// TIA Portal V17 export
// export: Created 2023-02-13T11:16:06.1178122Z, ExportSetting WithDefaults, DisplayName Totally Integrated Automation Portal, DisplayVersion V17, DisplayName TIA Portal Openness, DisplayVersion V17, DisplayName TIA Portal Teamcenter Gateway, DisplayVersion V17, DisplayName TIA Portal Version Control Interface, DisplayVersion V17, DisplayName SINAMICS Startdrive Advanced, DisplayVersion V17, DisplayName SINAMICS Startdrive G130, G150, S120, S150, SINAMICS MV, S210, DisplayVersion V17, DisplayName SINAMICS Startdrive G110M, G120, G120C, G120D, G120P, G115D, DisplayVersion V17, DisplayName STEP 7 Professional, DisplayVersion V17, DisplayName STEP 7 Safety, DisplayVersion V17, DisplayName WinCC Professional, DisplayVersion V17
DATA_BLOCK "CIP_Sto_to_CIP"   // DB191
{ S7_Optimized_Access := 'FALSE' }
VERSION : 0.1
// stored: AutoNumber false, DBAccessibleFromOPCUA true, DBAccessibleFromWebserver true, IsOnlyStoredInLoadMemory false, IsWriteProtectedInAS false
   VAR
      HeatBeat : Bool;
      CIP_Request : Bool;   // Cip Kitchen Ready
      ReturnPump_ON : Bool;   // Reqquest approved
      CIP_Complete : Bool;
      Valve_Line_Supply_Open : Bool;
      Spare : Bool;
      Spare_1 : Bool;
      Spare_2 : Bool;
      Spare_3 : Bool;
      Spare_4 : Bool;
      Spare_5 : Bool;
      Spare_6 : Bool;
      Spare_7 : Bool;
      Spare_8 : Bool;
      Spare_9 : Bool;
      Spare_10 : Bool;
      Data_Real : Real;
      Data_Real_1 : Real;
      Data_Real_2 : Real;
      Data_Real_3 : Real;
      Data_Real_4 : Real;
      Data_Real_5 : Real;
      Data_Real_6 : Real;
      Data_Real_7 : Real;
   END_VAR
BEGIN
END_DATA_BLOCK
